// TIA Portal V16 export
// export: Created 2023-03-29T11:03:22.5003153Z, ExportSetting WithDefaults, DisplayName Totally Integrated Automation Portal, DisplayVersion V16 Update 6, DisplayName TIA Portal Version Control Interface, DisplayVersion V16 Update 2, DisplayName TIA Portal Openness, DisplayVersion V16 Update 6, DisplayName STEP 7 Professional, DisplayVersion V16 Update 6, DisplayName STEP 7 Safety, DisplayVersion V16, DisplayName WinCC Advanced, DisplayVersion V16 Update 6
FUNCTION_BLOCK "godzinyPracy"   // FB19, LAD
{ S7_Optimized_Access := 'TRUE' }
AUTHOR : RTecmer
FAMILY : XMHour
VERSION : 0.1
// Licznik czasu pracy
// stored: AutoNumber true, IsIECCheckEnabled false, IsRetainMemResEnabled false, MemoryReserve 500, SetENOAutomatically false, UDAEnableTagReadback false
   VAR_INPUT
      Run_Device : Bool;
   END_VAR
   VAR_OUTPUT
      MW_hour : DWord;
      Sum_hour_sek : Real;   // Licznik sumator godzin i sekund na potrzeby wyznaczania dumchawy do pracy
   END_VAR
   VAR_IN_OUT
      Data_sek : Int;
      Reset { ExternalAccessible := 'False'; ExternalVisible := 'False'; ExternalWritable := 'False'} : Bool;
      Data_hour : DWord;
      Edge_Hz { ExternalAccessible := 'False'; ExternalVisible := 'False'; ExternalWritable := 'False'} : Bool;
   END_VAR
   VAR
      sek_real { ExternalAccessible := 'False'; ExternalVisible := 'False'; ExternalWritable := 'False'} : Real;   // pomocnicza konwerski sekund
      actSekReal { ExternalAccessible := 'False'; ExternalVisible := 'False'; ExternalWritable := 'False'} : Real;   // aktualne sekundy po konwersji
      hour_sek { ExternalAccessible := 'False'; ExternalVisible := 'False'; ExternalWritable := 'False'} : Real;
   END_VAR
   VAR_TEMP   // added for the SCL form of the ladder/FBD networks
      _w1 : Bool;
      _w2 : Bool;
   END_VAR
BEGIN

REGION Network 1
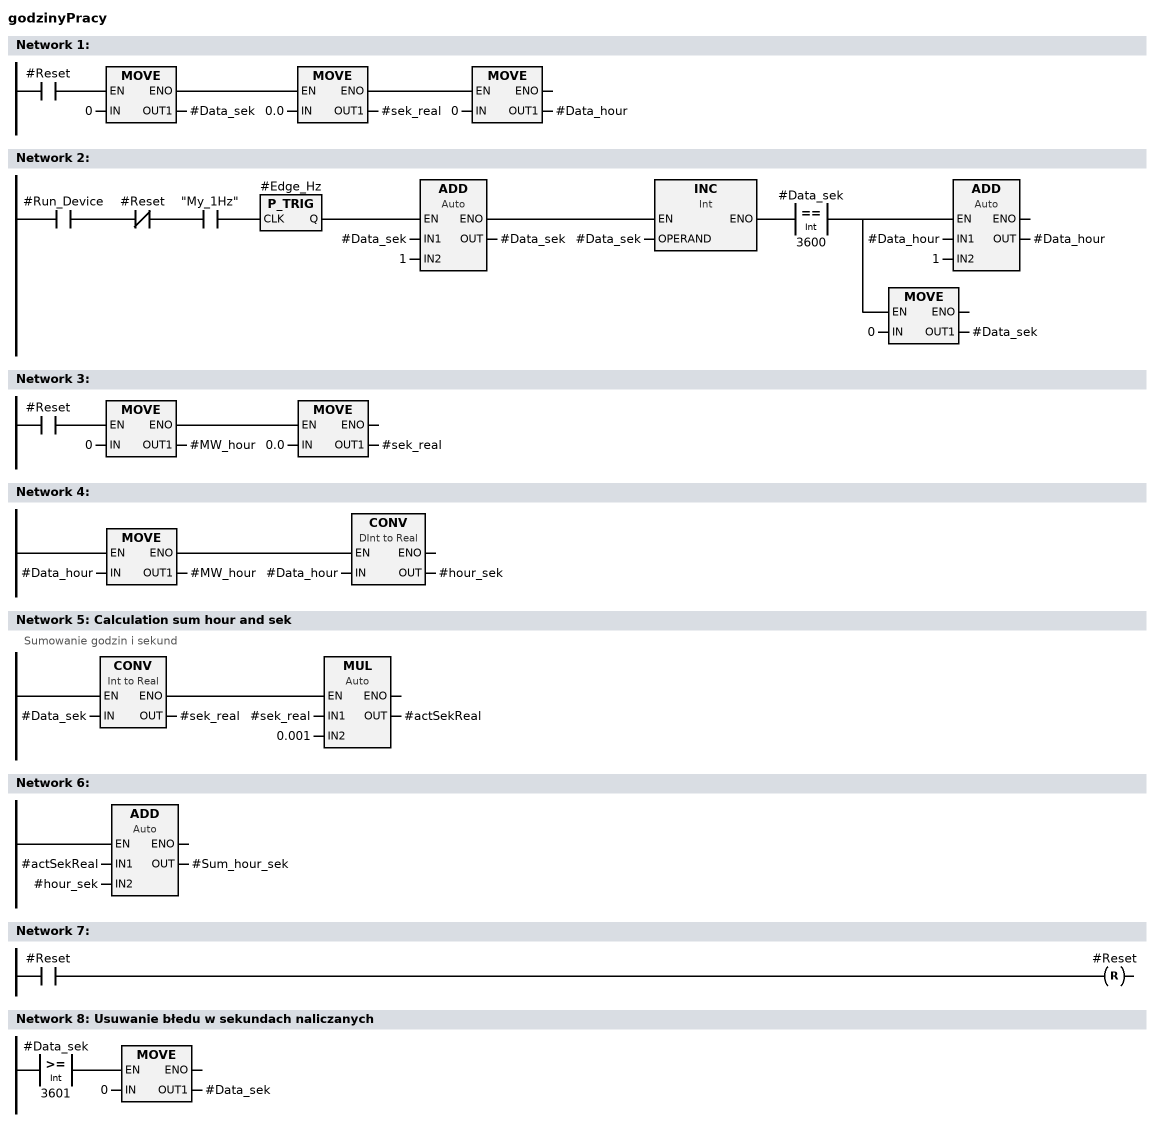
   RUNG wire#powerrail
      Contact( #Reset )
      { S7_GenerateENO := "TRUE" } Move(in := 0, out1 => #Data_sek)
      { S7_GenerateENO := "TRUE" } Move(in := 0.0, out1 => #sek_real)
      { S7_GenerateENO := "TRUE" } Move(in := 0, out1 => #Data_hour)
   END_RUNG
   // the same network as SCL:
   // ENO of a box is taken as its EN; it also drops when the box reports an error
   IF #Reset THEN
       #Data_sek := 0;
       #sek_real := 0.0;
       #Data_hour := 0;
   END_IF;
END_REGION

REGION Network 2
   RUNG wire#powerrail
      Contact( #Run_Device )
      I_Contact( #Reset )
      Contact( "My_1Hz" )
      P_Trig( #Edge_Hz )
      { S7_GenerateENO := "TRUE" } Add(in1 := #Data_sek, in2 := 1, out => #Data_sek)
      { S7_Templates := "DestType := Int"; S7_GenerateENO := "TRUE" } Inc( #Data_sek )
      { S7_Templates := "SrcType := Int" } EQ_Contact(in1 := #Data_sek, in2 := 3600)
      wire#w1
      { S7_GenerateENO := "TRUE" } Add(in1 := #Data_hour, in2 := 1, out => #Data_hour)
   END_RUNG
   RUNG wire#w1
      { S7_GenerateENO := "TRUE" } Move(in := 0, out1 => #Data_sek)
   END_RUNG
   // the same network as SCL:
   // ENO of a box is taken as its EN; it also drops when the box reports an error
   #_w1 := #Run_Device AND NOT #Reset AND "My_1Hz";
   #_w2 := #_w1 AND NOT #Edge_Hz;   // rising edge
   #Edge_Hz := #_w1;
   IF #_w2 THEN
       #Data_sek := #Data_sek + 1;
       #Data_sek := #Data_sek + 1;
   END_IF;
   IF #_w2 AND (#Data_sek = 3600) THEN
       #Data_hour := #Data_hour + 1;
       #Data_sek := 0;
   END_IF;
END_REGION

REGION Network 3
   RUNG wire#powerrail
      Contact( #Reset )
      { S7_GenerateENO := "TRUE" } Move(in := 0, out1 => #MW_hour)
      { S7_GenerateENO := "TRUE" } Move(in := 0.0, out1 => #sek_real)
   END_RUNG
   // the same network as SCL:
   // ENO of a box is taken as its EN; it also drops when the box reports an error
   IF #Reset THEN
       #MW_hour := 0;
       #sek_real := 0.0;
   END_IF;
END_REGION

REGION Network 4
   RUNG wire#powerrail
      { S7_GenerateENO := "TRUE" } Move(in := #Data_hour, out1 => #MW_hour)
      { S7_Templates := "[SrcType := DInt, DestType := Real]" } Convert(in := #Data_hour, out => #hour_sek)
   END_RUNG
   // the same network as SCL:
   // ENO of a box is taken as its EN; it also drops when the box reports an error
   #MW_hour := #Data_hour;
   #hour_sek := DINT_TO_REAL(#Data_hour);
END_REGION

REGION Network 5: Calculation sum hour and sek
   // Sumowanie godzin i sekund
   RUNG wire#powerrail
      { S7_Templates := "[SrcType := Int, DestType := Real]" } Convert(in := #Data_sek, out => #sek_real)
      Mul(in1 := #sek_real, in2 := 0.001, out => #actSekReal)
   END_RUNG
   // the same network as SCL:
   #sek_real := INT_TO_REAL(#Data_sek);
   #actSekReal := #sek_real * 0.001;
END_REGION

REGION Network 6
   RUNG wire#powerrail
      Add(in1 := #actSekReal, in2 := #hour_sek, out => #Sum_hour_sek)
   END_RUNG
   // the same network as SCL:
   #Sum_hour_sek := #actSekReal + #hour_sek;
END_REGION

REGION Network 7
   RUNG wire#powerrail
      Contact( #Reset )
      R_Coil( #Reset )
   END_RUNG
   // the same network as SCL:
   IF #Reset THEN #Reset := FALSE; END_IF;
END_REGION

REGION Network 8: Usuwanie błedu w sekundach naliczanych
   RUNG wire#powerrail
      { S7_Templates := "SrcType := Int" } GE_Contact(in1 := #Data_sek, in2 := 3601)
      { S7_GenerateENO := "TRUE" } Move(in := 0, out1 => #Data_sek)
   END_RUNG
   // the same network as SCL:
   IF #Data_sek >= 3601 THEN #Data_sek := 0; END_IF;
END_REGION
END_FUNCTION_BLOCK
